{attribute 'global_init_slot' := '49991'}
{attribute 'qualified_only'}
VAR_GLOBAL CONSTANT
	// encoder resolution
	g_incEncoderRes :ARRAY[1..g_sJntNum] OF DINT :=[8(65536)];
	g_absEncoderRes :ARRAY[1..g_sJntNum] OF DINT :=[8(16777216)];
	
	// reduction ratio
	g_motorReduction :ARRAY[1..g_sJntNum] OF LREAL :=[ 81,81,  (66.0/10)*2*pi/0.010, 5(388125.0/4693)];
	g_absEncoderReduction :ARRAY[1..g_sJntNum] OF LREAL :=[2(1.0), 2*PI/0.64, 5(1.0)];
	
	// motor parameters
	g_motorTrqConst :ARRAY[1..g_sJntNum] OF LREAL :=[ 0.16,0.16, 0.017,5(0.0193)];
	g_motorMaxCurrent :ARRAY[1..g_sJntNum] OF LREAL :=[ 5600,5600,  500, 5(500)];//mA
	
	// motor encoder direction
	g_motorDir :ARRAY[1..g_sJntNum] OF INT :=[-1, 1, -1, 1, 1, 1, 1, 1];
																 
	// joint position limit
	g_minJntPos: ARRAY[1..g_sJntNum] OF LREAL:=[-pi,	-pi/2,	0.15, 	5(-99*pi)];	
	g_maxJntPos: ARRAY[1..g_sJntNum] OF LREAL:=[pi,	1.196, 	0.58, 		5(99*pi)];
	
	// joint velocity limit
	g_maxJntVel :ARRAY[1..g_sJntNum] OF LREAL :=[1.2, 1.2, 0.2, 5(2*pi)];
	
	// joint SDO address
	g_slaveArmNetID: ARRAY[1..4] OF T_AmsNetId:=['169.254.240.177.5.1','169.254.223.239.7.1','169.254.223.239.9.1','169.254.223.239.10.1'];
	g_slaveJointNetPort:ARRAY[1..g_sArmNum,1..g_sJntNum] OF UINT :=[
		1004,	1005,	1006,	2(1007),	3(1008),
		1006,	1007,	1008,	2(1009),	3(1010),
		1006,	1007,	1008,	2(1009),	3(1010),
		1006,	1007,	1008,	2(1009),	3(1010)];
		
END_VAR

(* stored: Version 1.1.0.1, ProductVersion 3.1.4024.11
   GVL GVL_SlaveMotorParameters: Id {cf487053-15bb-46bd-a4ed-bbb1df690beb} *)
